PROGRAM p07_memoryCell
VAR
	S0: BOOL;
	S1: BOOL;
	L0: BOOL;
	L1: BOOL;
	L2: BOOL;
	RS_cell: RS;
	SR_cell: SR;
END_VAR

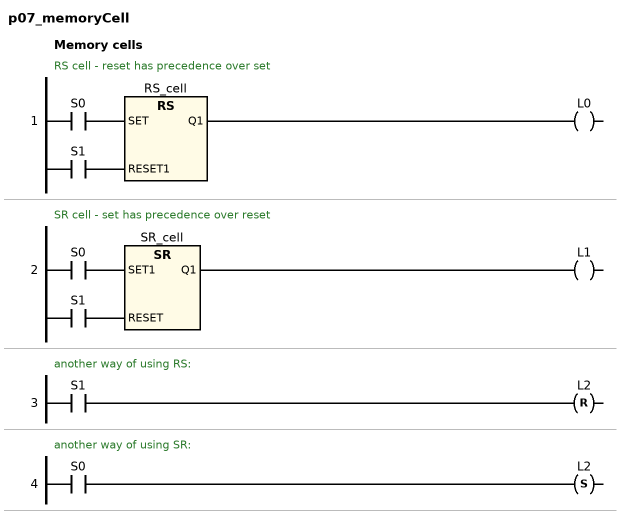
// NETWORK 1: Memory cells
// RS cell - reset has precedence over set
RS_cell(SET := S0, RESET1 := S1); // RS
L0 := RS_cell.Q1;

// NETWORK 2
// SR cell - set has precedence over reset
SR_cell(SET1 := S0, RESET := S1); // SR
L1 := SR_cell.Q1;

// NETWORK 3
// another way of using RS:
L2 R= S1;

// NETWORK 4
// another way of using SR:
L2 S= S0;

END_PROGRAM

(* stored: Version 1.1.0.1, ProductVersion 3.1.4024.13
   POU p07_memoryCell: Id {ce0d3116-9483-44f7-b54e-7ccbe8a72c18}, SpecialFunc None *)
